{attribute addProperty BoxType "EL9221-4030-0018"}
{attribute addProperty Id "OCP_InputsAT %I*OCP_Inputs_FE08AF3C3240OCP_OutputsAT %Q*OCP_Outputs_F330A9161620WcStateAT %I*WcState_F855686C1620InfoDataAT %I*InfoData_BC63D37F80100"}
{attribute addProperty CRC "4286454698"}
{attribute addProperty SizeInBites "144"}
{attribute addProperty SizeInBytes "18"}
TYPE EL9221_0E818766 :
STRUCT
	{attribute addProperty Name "OCP_Inputs"}
	OCP_Inputs : OCP_Inputs_FE08AF3C;
	{attribute addProperty Name "OCP_Outputs"}
	OCP_Outputs : OCP_Outputs_F330A916;
	{attribute addProperty Name "WcState"}
	WcState : WcState_F855686C;
	{attribute addProperty Name "InfoData"}
	InfoData : InfoData_BC63D37F;
END_STRUCT
END_TYPE

(* stored: Version 1.2.0.0, ProductVersion 3.1.4024.9
   DUT EL9221_0E818766: Id {4e1ae38f-1dc6-4ccb-8d98-ea10247e09e6} *)
